FUNCTION alg_M_Distributing_atpos : ARRAY[0..2] OF BOOL
VAR_INPUT
	state: STATE;
END_VAR

alg_M_Distributing_atpos := makeArray1(ivar_s_xpos_at1, ivar_s_xpos_at2, ivar_s_xpos_at3);

END_FUNCTION

(* stored: Version 1.1.0.1, ProductVersion 3.1.4022.18
   POU alg_M_Distributing_atpos: Id {3c0c0c6a-d9eb-431b-8f1a-8c7dd2a2de8d}, SpecialFunc None *)
